Fanuc KAREL source: kt00106.KL

-- PROVISIONAL review KL for V940-1; original PC SHA256 b74b6d271c0def70f751349019f9920fcfaebc8f3e76c7e0a492140179ed10bd
-- Incomplete behavior may be omitted. Consult companion uncertainty JSON. Do not deploy.
PROGRAM KT00106
%NOLOCKGROUP
VAR
  R1 : REAL
  I2 : INTEGER
  OUT : REAL
BEGIN
  -- V9_ZERO_TABLE_METADATA_HINT layout=0001; no indexed target words; source/name/runtime held
  -- UNRESOLVED_PC offsets 5-16; opcodes 2E,23
  -- UNRESOLVED_PC offsets 21-32; opcodes 2E,23
  -- UNRESOLVED_PC offsets 37-57; opcodes 21,21,64,6C,23
  -- UNRESOLVED_PC offsets 62-66; opcodes 7F
END KT00106
